INTERFACE I_DataSource

METHOD Call : BOOL
END_METHOD

METHOD GetData : BOOL
VAR_INPUT
	nElement: UDINT;
END_VAR
END_METHOD

METHOD HistoricalCtrl : BOOL
VAR_INPUT
	stCtrl: REFERENCE TO ST_HMI_DataSourceCtrl;
	stHistStreamInfo: REFERENCE TO ST_HMI_DataSourceHist;
	stRecordInfo: REFERENCE TO ST_HMI_DataSourceHistRecordInfo;
END_VAR
END_METHOD

METHOD UpdateRecordList : BOOL
VAR_INPUT
	stCtrl: REFERENCE TO ST_HMI_DataSourceCtrl;
	sStreamSystemID: GUID;
	stHistStreamInfo: REFERENCE TO ST_HMI_DataSourceHist;
END_VAR
END_METHOD

METHOD NewDataAvailable : BOOL
VAR_INPUT
	nLastDataHandle: ULINT;
END_VAR
END_METHOD

PROPERTY nDataHandle : ULINT
GET
END_GET
END_PROPERTY

PROPERTY nElements : UDINT
GET
END_GET
END_PROPERTY

PROPERTY dtTimestamp : DCTIMESTRUCT
GET
END_GET
END_PROPERTY

END_INTERFACE

(* stored: Version 1.1.0.1
   Itf I_DataSource: Id 5731df2d-e237-423e-b0c2-7e323003ce67
   Method Call: Id 681153a6-1fc8-4130-8dfc-b5dca248a96e
   Method GetData: Id 75d4352d-ddbe-42d6-a606-dcfab603fe7c
   Method HistoricalCtrl: Id b9b03f21-462c-4537-a463-e7fcea413b3c
   Method UpdateRecordList: Id d5019b04-da63-4b13-b02c-054ea6d34cfe
   Method NewDataAvailable: Id bb8b9e8f-7426-42c5-b967-b4fcb2e1ccfe
   Property nDataHandle: Id bcb14690-650c-4ccd-91a1-bd61abd77a54
   Get Get: Id e4070158-09b5-40c6-9098-a01bdbee2773
   Property nElements: Id f8f7340c-ca41-4f9c-b710-d17cad606579
   Get Get: Id ff96fdbe-217d-45b4-8ef3-8ab2a224cf29
   Property dtTimestamp: Id 670c7b46-bbc1-40c0-b758-42d0cdb415f0
   Get Get: Id 85e98876-2f50-40e4-8571-99f9acaaa438 *)
